INTERFACE I_AxisBase EXTENDS I_Cyclic

METHOD PUBLIC DisableAxis : HRESULT
VAR_INPUT
END_VAR
END_METHOD

METHOD PUBLIC EnableAxis : HRESULT
VAR_INPUT
END_VAR
END_METHOD

METHOD GetErrorId : DWORD
VAR_INPUT
END_VAR
END_METHOD

METHOD PUBLIC HaltAxis : HRESULT
VAR
END_VAR
END_METHOD

METHOD hasError : BOOL
VAR_INPUT
END_VAR
END_METHOD

METHOD isEnabled : BOOL
VAR_INPUT
END_VAR
END_METHOD

METHOD PUBLIC Reset : HRESULT
VAR
END_VAR
END_METHOD

END_INTERFACE

(* stored: Version 1.1.0.1
   Itf I_AxisBase: Id {0ef07e09-d612-4b35-8507-c5527a9d7e82}
   Method DisableAxis: Id {9aa78aa4-6937-4925-a0b3-e6b55191b9b8}
   Method EnableAxis: Id {1d051842-9ad9-43b4-9c63-942a1b02943c}
   Method GetErrorId: Id {0e102596-72b8-4e67-b2e5-ef82f66c692e}
   Method HaltAxis: Id {f00a986d-e8a1-4ddc-8d6f-7dfd0ff96b72}
   Method hasError: Id {b463ab8b-6f68-4ef7-aee6-f909cd031bdf}
   Method isEnabled: Id {74def401-5519-4834-a231-64b141cc4fba}
   Method Reset: Id {70c30306-2843-45ea-9390-dee5671086b2} *)
